FUNCTION_BLOCK Q_ObjSelectInput (* Command Select input object ( Part 6 - F.6 ) *)
  (* Standard: ISO 11783-6; Description: This command is used to force the selection of an input field object. Return values iso_s16 - E_NO_ERR - OK - E_OVERFLOW - buffer overflow - E_NOACT - Command not possible in current state - E_NO_INSTANCE - No VT client available *)
  (* Version 1.0, 2022-07-08, franz *)
  (* Documentation:
  This command is used to force the selection of an input field object.
   Return values
   iso_s16
    - E_NO_ERR - OK
   - E_OVERFLOW - buffer overflow
   - E_NOACT - Command not possible in current state
   - E_NO_INSTANCE - No VT client available
  *)
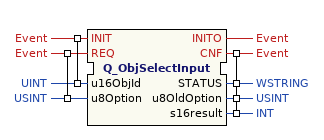
  EVENT_INPUT
    INIT WITH u16ObjId; (* Service Initialization *)
    REQ WITH u8Option; (* Service Request *)
  END_EVENT
  EVENT_OUTPUT
    INITO; (* Initialization Confirm *)
    CNF WITH STATUS, s16result, u8OldOption; (* Confirmation of Requested Service *)
  END_EVENT
  VAR_INPUT
    u16ObjId : UINT; (* Object ID *)
    u8Option : USINT; (* normal: 0xFF, for Version 4 also 0 possible *)
  END_VAR
  VAR_OUTPUT
    STATUS : WSTRING; (* Service Status *)
    u8OldOption : USINT; (* Old normal: 0xFF, for Version 4 also 0 possible *)
    s16result : INT; (* retval see description *)
  END_VAR
END_FUNCTION_BLOCK
